TYPE ASCF_CC_OPCUACS_ScheduleDataType1:
STRUCT
	Reader		: BOOL					:= TRUE;
	Writer		: BOOL					:= FALSE;
	NextID		: INT					:= 1;
	Schedule	: ARRAY[0..0] OF INT	:= [0];
END_STRUCT
END_TYPE

(* stored: Version 1.1.0.1, ProductVersion 3.1.4026.4
   DUT ASCF_CC_OPCUACS_ScheduleDataType1: Id {af0c4982-29aa-415d-949f-6effaae409d0} *)
